{attribute 'qualified_only'}
//{attribute 'strict'}
{attribute 'to_string'}
TYPE E_PROGRESS :
(
  // progress is used in project to mirror state of requested command/function
  INVALID,
  INIT,
	BUSY          :=  100,
  STARTUP       :=  200,
  PREPARE       :=  300,
  READY         :=  400,
  WAITING       :=  500,
  WORKING       :=  600,

  DONE          := 1000,

  ERROR         := 9000

)UINT;
END_TYPE

(* stored: Version 1.1.0.1, ProductVersion 3.1.4024.12
   DUT E_PROGRESS: Id {01ea6048-5c71-0a1f-04ff-ba0b7cf1e485} *)
